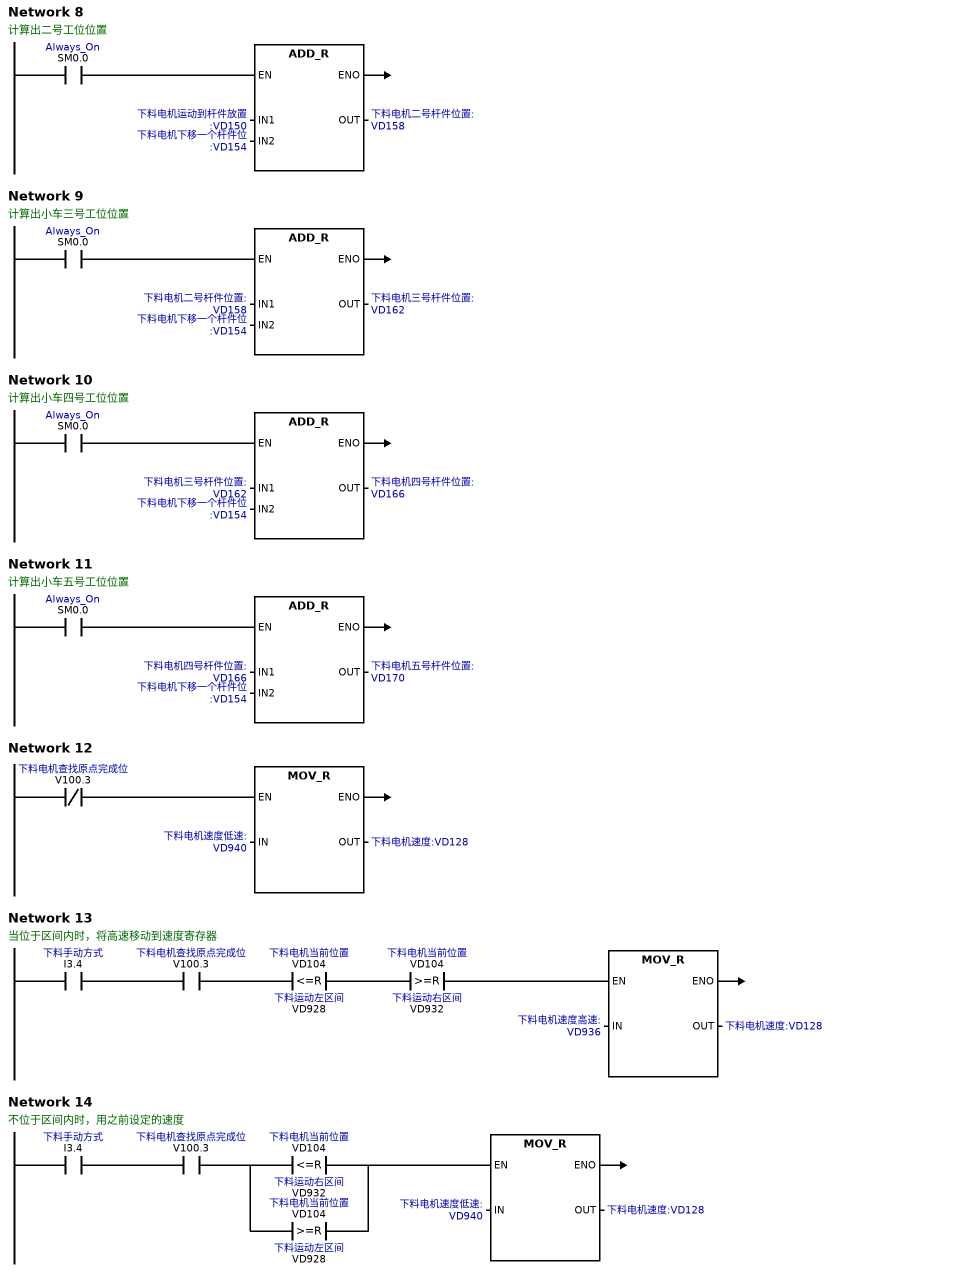
[picture p24: SBR15 networks 8-14]
Network 8
// 计算出二号工位位置
LD     Always_On:SM0.0
MOVR   下料电机运动到杆件放置:VD150, 下料电机二号杆件位置:VD158
+R     下料电机下移一个杆件位:VD154, 下料电机二号杆件位置:VD158
Network 9
// 计算出小车三号工位位置
LD     Always_On:SM0.0
MOVR   下料电机二号杆件位置:VD158, 下料电机三号杆件位置:VD162
+R     下料电机下移一个杆件位:VD154, 下料电机三号杆件位置:VD162
Network 10
// 计算出小车四号工位位置
LD     Always_On:SM0.0
MOVR   下料电机三号杆件位置:VD162, 下料电机四号杆件位置:VD166
+R     下料电机下移一个杆件位:VD154, 下料电机四号杆件位置:VD166
Network 11
// 计算出小车五号工位位置
LD     Always_On:SM0.0
MOVR   下料电机四号杆件位置:VD166, 下料电机五号杆件位置:VD170
+R     下料电机下移一个杆件位:VD154, 下料电机五号杆件位置:VD170
Network 12
LDN    下料电机查找原点完成位:V100.3
MOVR   下料电机速度低速:VD940, 下料电机速度:VD128
Network 13
// 当位于区间内时，将高速移动到速度寄存器
LD     下料手动方式:I3.4
A      下料电机查找原点完成位:V100.3
AR<=   下料电机当前位置:VD104, 下料运动左区间:VD928
AR>=   下料电机当前位置:VD104, 下料运动右区间:VD932
MOVR   下料电机速度高速:VD936, 下料电机速度:VD128
Network 14
// 不位于区间内时，用之前设定的速度
LD     下料手动方式:I3.4
A      下料电机查找原点完成位:V100.3
LDR<=  下料电机当前位置:VD104, 下料运动右区间:VD932
OR>=   下料电机当前位置:VD104, 下料运动左区间:VD928
ALD
MOVR   下料电机速度低速:VD940, 下料电机速度:VD128
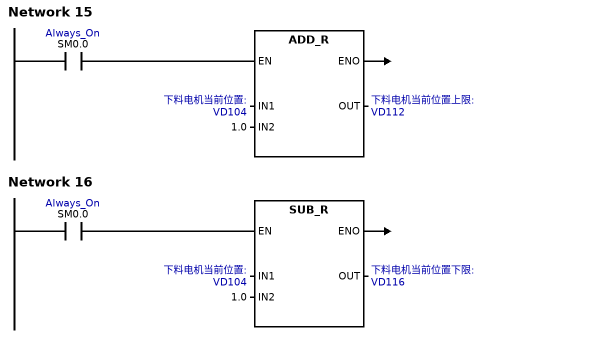
Network 15
LD     Always_On:SM0.0
MOVR   下料电机当前位置:VD104, 下料电机当前位置上限:VD112
+R     1.0, 下料电机当前位置上限:VD112
Network 16
LD     Always_On:SM0.0
MOVR   下料电机当前位置:VD104, 下料电机当前位置下限:VD116
-R     1.0, 下料电机当前位置下限:VD116
END_SUBROUTINE_BLOCK

SUBROUTINE_BLOCK 冷却初始化:SBR16
TITLE=子程序注释
BEGIN
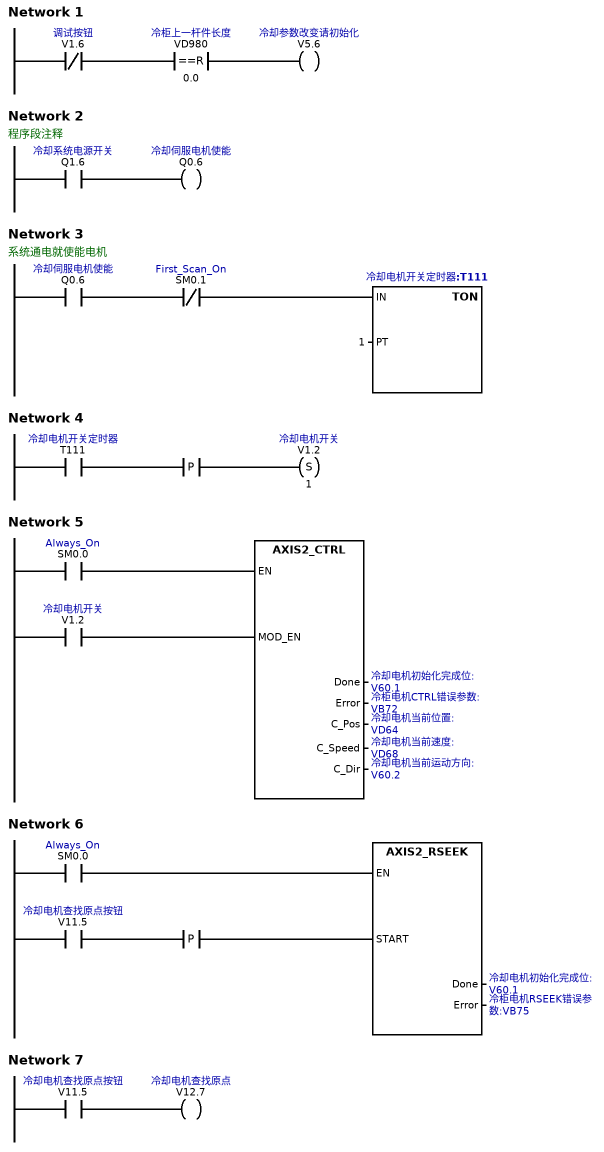
Network 1
LDN    调试按钮:V1.6
AR=    冷柜上一杆件长度:VD980, 0.0
=      冷却参数改变请初始化:V5.6
Network 2
// 程序段注释
LD     冷却系统电源开关:Q1.6
=      冷却伺服电机使能:Q0.6
Network 3
// 系统通电就使能电机
LD     冷却伺服电机使能:Q0.6
AN     First_Scan_On:SM0.1
TON    冷却电机开关定时器:T111, 1
Network 4
LD     冷却电机开关定时器:T111
EU
S      冷却电机开关:V1.2, 1
Network 5
LD     Always_On:SM0.0
=      L60.0
LD     冷却电机开关:V1.2
=      L63.7
LD     L60.0
CALL   AXIS2_CTRL:SBR10, L63.7, 冷却电机初始化完成位:V60.1, 冷柜电机CTRL错误参数:VB72, 冷却电机当前位置:VD64, 冷却电机当前速度:VD68, 冷却电机当前运动方向:V60.2
Network 6
LD     Always_On:SM0.0
=      L60.0
LD     冷却电机查找原点按钮:V11.5
EU
=      L63.7
LD     L60.0
CALL   AXIS2_RSEEK:SBR13, L63.7, 冷却电机初始化完成位:V60.1, 冷柜电机RSEEK错误参数:VB75
Network 7
LD     冷却电机查找原点按钮:V11.5
=      冷却电机查找原点:V12.7
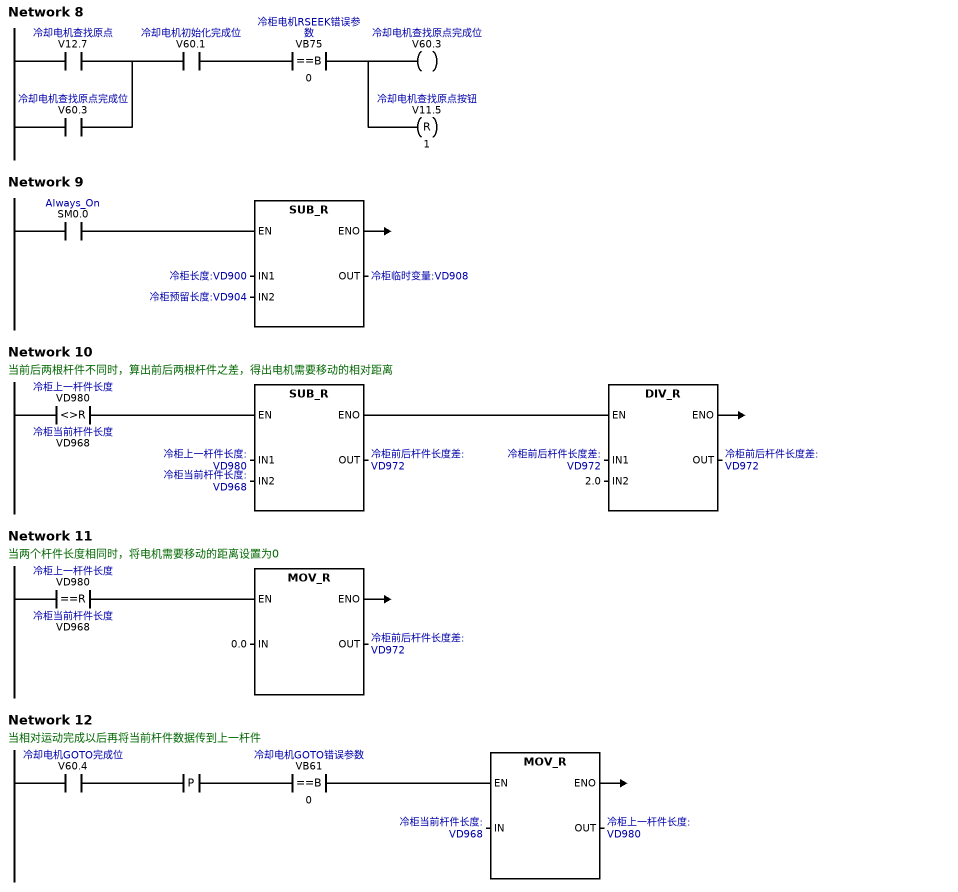
Network 8
LD     冷却电机查找原点:V12.7
O      冷却电机查找原点完成位:V60.3
A      冷却电机初始化完成位:V60.1
AB=    冷柜电机RSEEK错误参数:VB75, 0
=      冷却电机查找原点完成位:V60.3
R      冷却电机查找原点按钮:V11.5, 1
Network 9
LD     Always_On:SM0.0
MOVR   冷柜长度:VD900, 冷柜临时变量:VD908
-R     冷柜预留长度:VD904, 冷柜临时变量:VD908
Network 10
// 当前后两根杆件不同时，算出前后两根杆件之差，得出电机需要移动的相对距离
LDR<>  冷柜上一杆件长度:VD980, 冷柜当前杆件长度:VD968
MOVR   冷柜上一杆件长度:VD980, 冷柜前后杆件长度差:VD972
AENO
-R     冷柜当前杆件长度:VD968, 冷柜前后杆件长度差:VD972
AENO
/R     2.0, 冷柜前后杆件长度差:VD972
Network 11
// 当两个杆件长度相同时，将电机需要移动的距离设置为0
LDR=   冷柜上一杆件长度:VD980, 冷柜当前杆件长度:VD968
MOVR   0.0, 冷柜前后杆件长度差:VD972
Network 12
// 当相对运动完成以后再将当前杆件数据传到上一杆件
LD     冷却电机GOTO完成位:V60.4
EU
AB=    冷却电机GOTO错误参数:VB61, 0
MOVR   冷柜当前杆件长度:VD968, 冷柜上一杆件长度:VD980
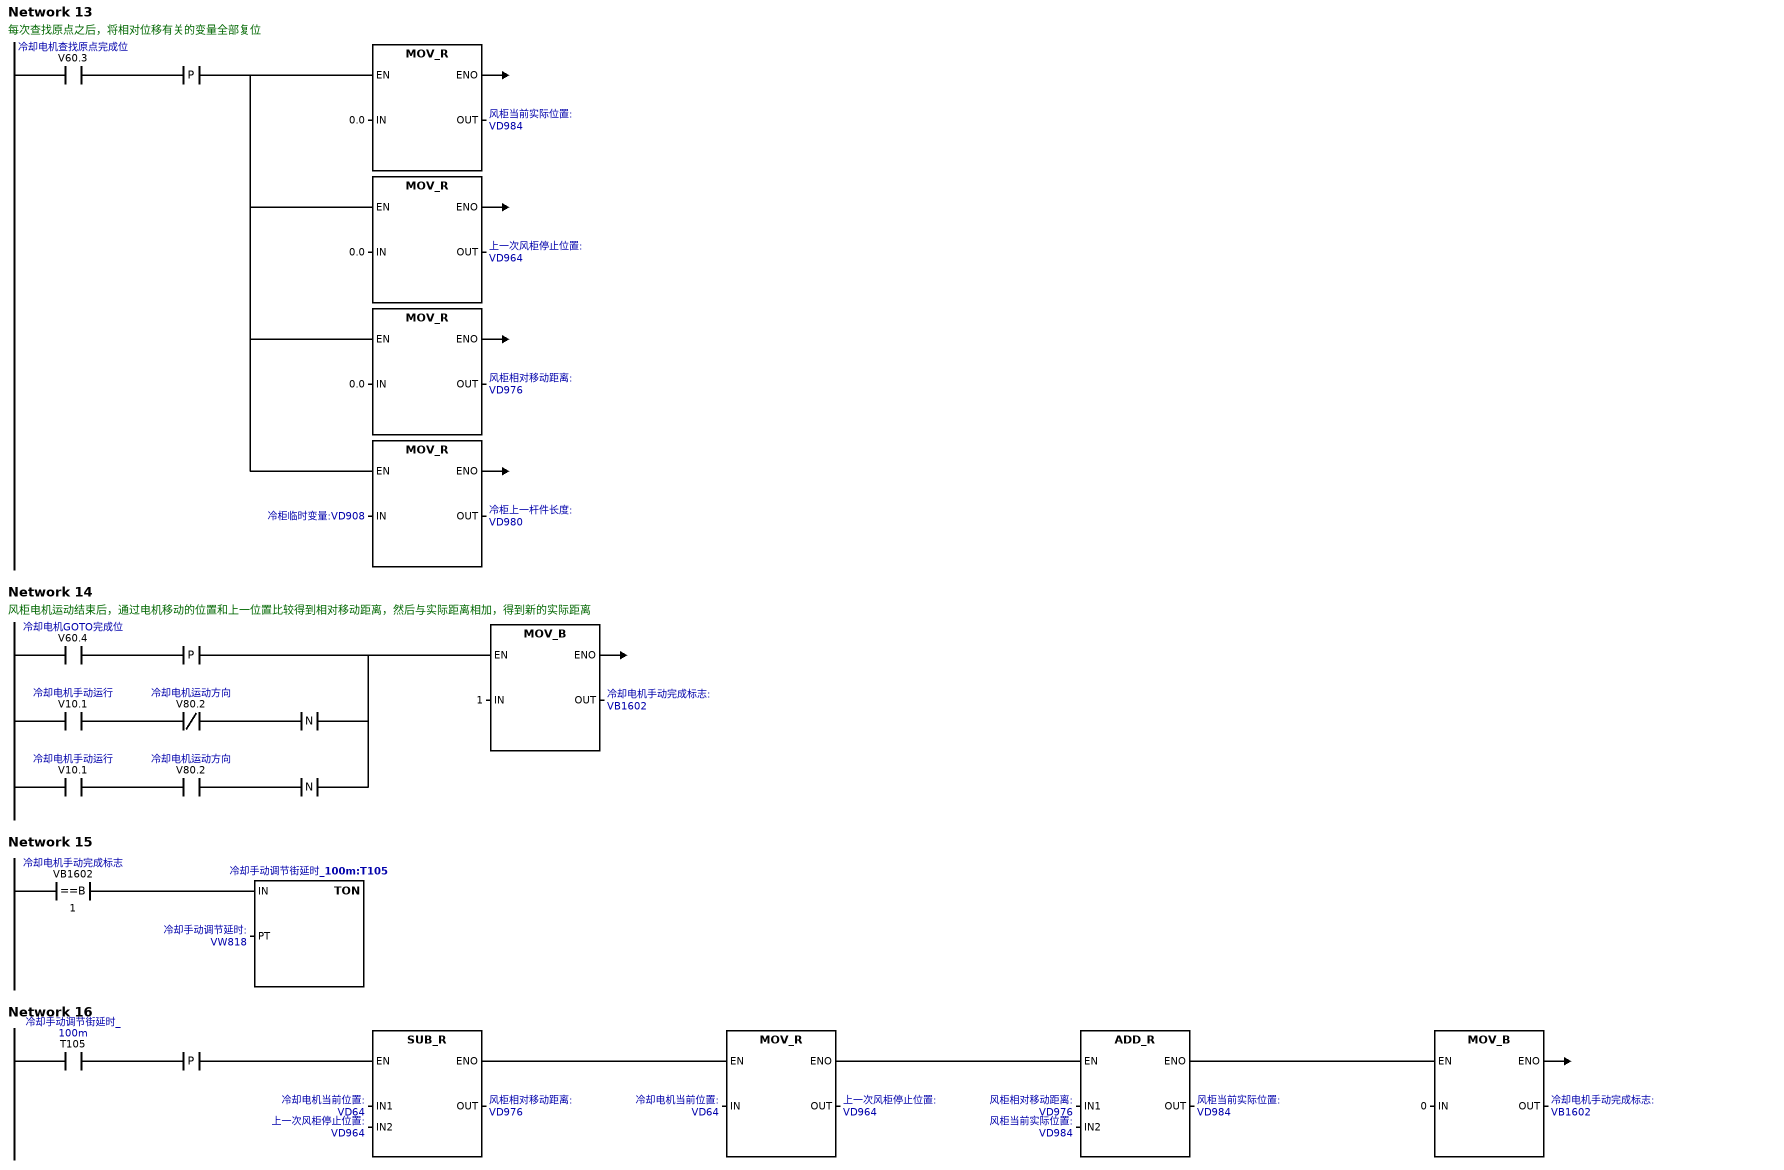
Network 13
// 每次查找原点之后，将相对位移有关的变量全部复位
LD     冷却电机查找原点完成位:V60.3
EU
MOVR   0.0, 风柜当前实际位置:VD984
MOVR   0.0, 上一次风柜停止位置:VD964
MOVR   0.0, 风柜相对移动距离:VD976
MOVR   冷柜临时变量:VD908, 冷柜上一杆件长度:VD980
Network 14
// 风柜电机运动结束后，通过电机移动的位置和上一位置比较得到相对移动距离，然后与实际距离相加，得到新的实际距离
LD     冷却电机GOTO完成位:V60.4
EU
LD     冷却电机手动运行:V10.1
AN     冷却电机运动方向:V80.2
ED
OLD
LD     冷却电机手动运行:V10.1
A      冷却电机运动方向:V80.2
ED
OLD
MOVB   1, 冷却电机手动完成标志:VB1602
Network 15
LDB=   冷却电机手动完成标志:VB1602, 1
TON    冷却手动调节街延时_100m:T105, 冷却手动调节延时:VW818
Network 16
LD     冷却手动调节街延时_100m:T105
EU
MOVR   冷却电机当前位置:VD64, 风柜相对移动距离:VD976
AENO
-R     上一次风柜停止位置:VD964, 风柜相对移动距离:VD976
AENO
MOVR   冷却电机当前位置:VD64, 上一次风柜停止位置:VD964
AENO
+R     风柜相对移动距离:VD976, 风柜当前实际位置:VD984
AENO
MOVB   0, 冷却电机手动完成标志:VB1602
END_SUBROUTINE_BLOCK

SUBROUTINE_BLOCK 上料选号:SBR17
TITLE=子程序注释
BEGIN
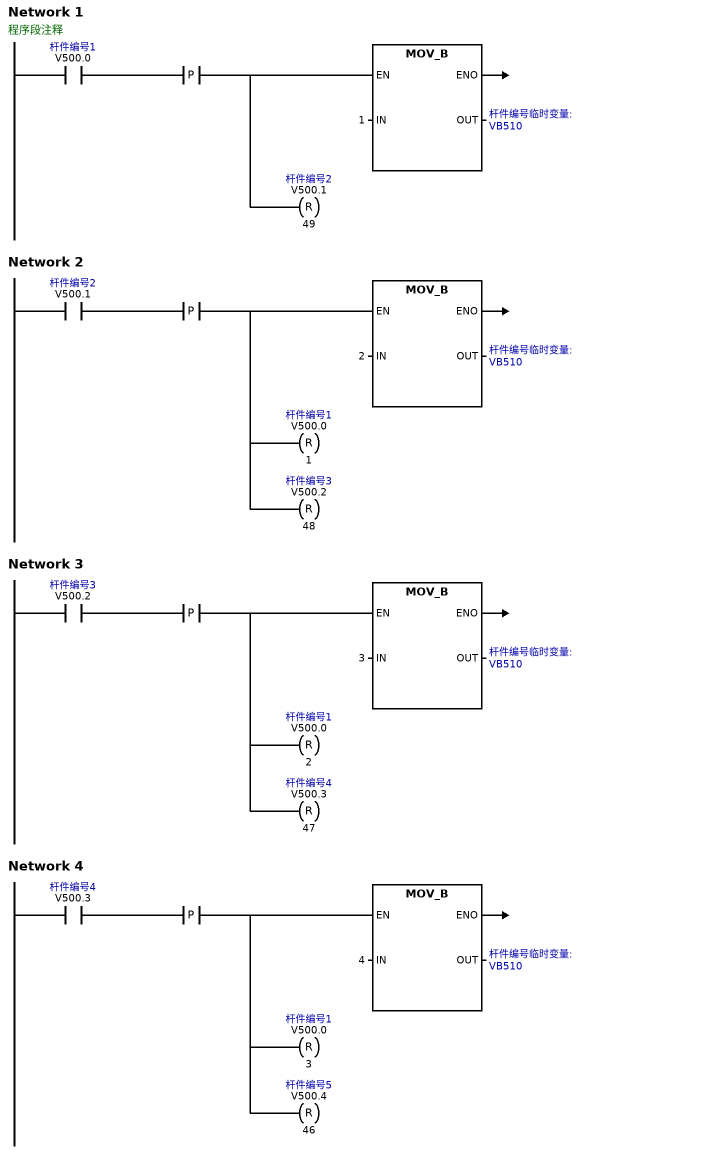
Network 1
// 程序段注释
LD     杆件编号1:V500.0
EU
MOVB   1, 杆件编号临时变量:VB510
R      杆件编号2:V500.1, 49
Network 2
LD     杆件编号2:V500.1
EU
MOVB   2, 杆件编号临时变量:VB510
R      杆件编号1:V500.0, 1
R      杆件编号3:V500.2, 48
Network 3
LD     杆件编号3:V500.2
EU
MOVB   3, 杆件编号临时变量:VB510
R      杆件编号1:V500.0, 2
R      杆件编号4:V500.3, 47
Network 4
LD     杆件编号4:V500.3
EU
MOVB   4, 杆件编号临时变量:VB510
R      杆件编号1:V500.0, 3
R      杆件编号5:V500.4, 46
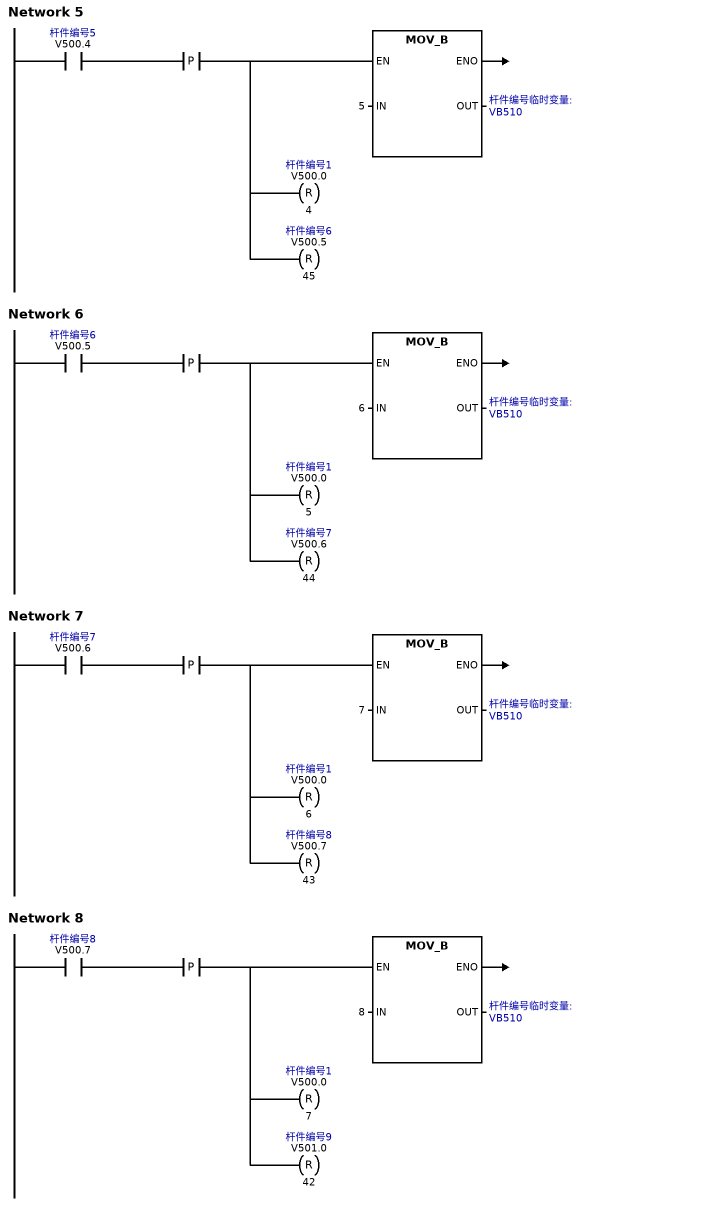
Network 5
LD     杆件编号5:V500.4
EU
MOVB   5, 杆件编号临时变量:VB510
R      杆件编号1:V500.0, 4
R      杆件编号6:V500.5, 45
Network 6
LD     杆件编号6:V500.5
EU
MOVB   6, 杆件编号临时变量:VB510
R      杆件编号1:V500.0, 5
R      杆件编号7:V500.6, 44
Network 7
LD     杆件编号7:V500.6
EU
MOVB   7, 杆件编号临时变量:VB510
R      杆件编号1:V500.0, 6
R      杆件编号8:V500.7, 43
Network 8
LD     杆件编号8:V500.7
EU
MOVB   8, 杆件编号临时变量:VB510
R      杆件编号1:V500.0, 7
R      杆件编号9:V501.0, 42
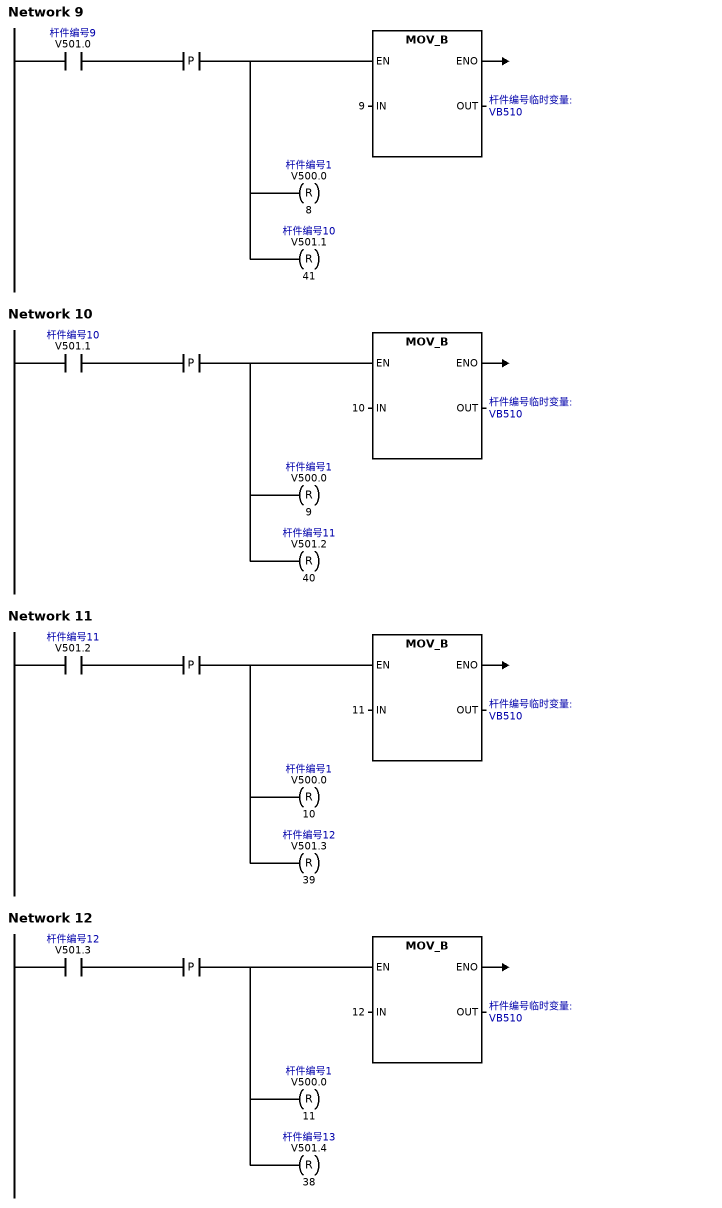
Network 9
LD     杆件编号9:V501.0
EU
MOVB   9, 杆件编号临时变量:VB510
R      杆件编号1:V500.0, 8
R      杆件编号10:V501.1, 41
Network 10
LD     杆件编号10:V501.1
EU
MOVB   10, 杆件编号临时变量:VB510
R      杆件编号1:V500.0, 9
R      杆件编号11:V501.2, 40
Network 11
LD     杆件编号11:V501.2
EU
MOVB   11, 杆件编号临时变量:VB510
R      杆件编号1:V500.0, 10
R      杆件编号12:V501.3, 39
Network 12
LD     杆件编号12:V501.3
EU
MOVB   12, 杆件编号临时变量:VB510
R      杆件编号1:V500.0, 11
R      杆件编号13:V501.4, 38
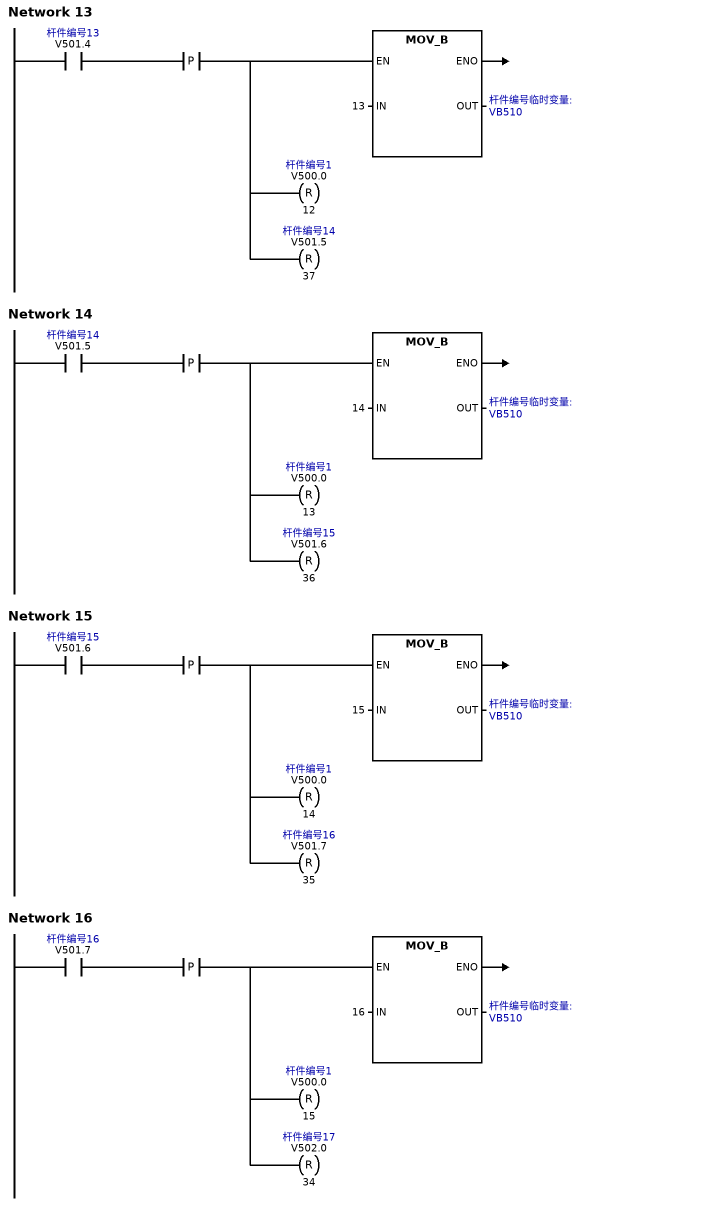
Network 13
LD     杆件编号13:V501.4
EU
MOVB   13, 杆件编号临时变量:VB510
R      杆件编号1:V500.0, 12
R      杆件编号14:V501.5, 37
Network 14
LD     杆件编号14:V501.5
EU
MOVB   14, 杆件编号临时变量:VB510
R      杆件编号1:V500.0, 13
R      杆件编号15:V501.6, 36
Network 15
LD     杆件编号15:V501.6
EU
MOVB   15, 杆件编号临时变量:VB510
R      杆件编号1:V500.0, 14
R      杆件编号16:V501.7, 35
Network 16
LD     杆件编号16:V501.7
EU
MOVB   16, 杆件编号临时变量:VB510
R      杆件编号1:V500.0, 15
R      杆件编号17:V502.0, 34
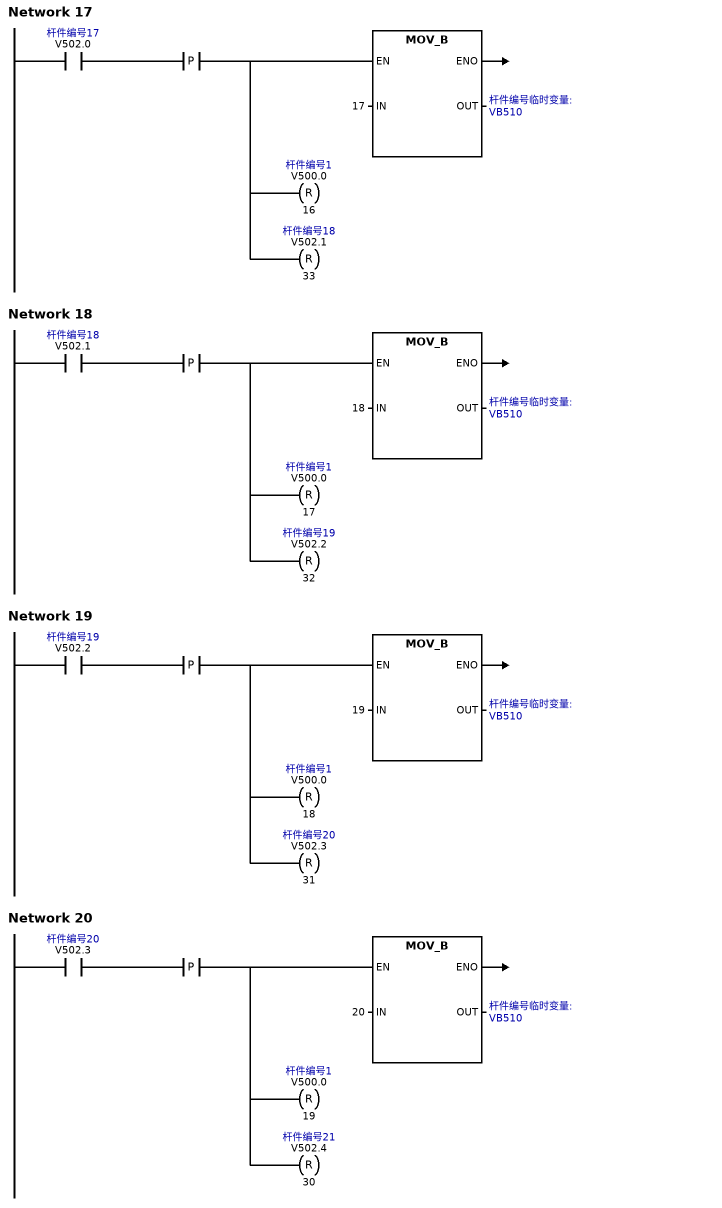
Network 17
LD     杆件编号17:V502.0
EU
MOVB   17, 杆件编号临时变量:VB510
R      杆件编号1:V500.0, 16
R      杆件编号18:V502.1, 33
Network 18
LD     杆件编号18:V502.1
EU
MOVB   18, 杆件编号临时变量:VB510
R      杆件编号1:V500.0, 17
R      杆件编号19:V502.2, 32
Network 19
LD     杆件编号19:V502.2
EU
MOVB   19, 杆件编号临时变量:VB510
R      杆件编号1:V500.0, 18
R      杆件编号20:V502.3, 31
Network 20
LD     杆件编号20:V502.3
EU
MOVB   20, 杆件编号临时变量:VB510
R      杆件编号1:V500.0, 19
R      杆件编号21:V502.4, 30
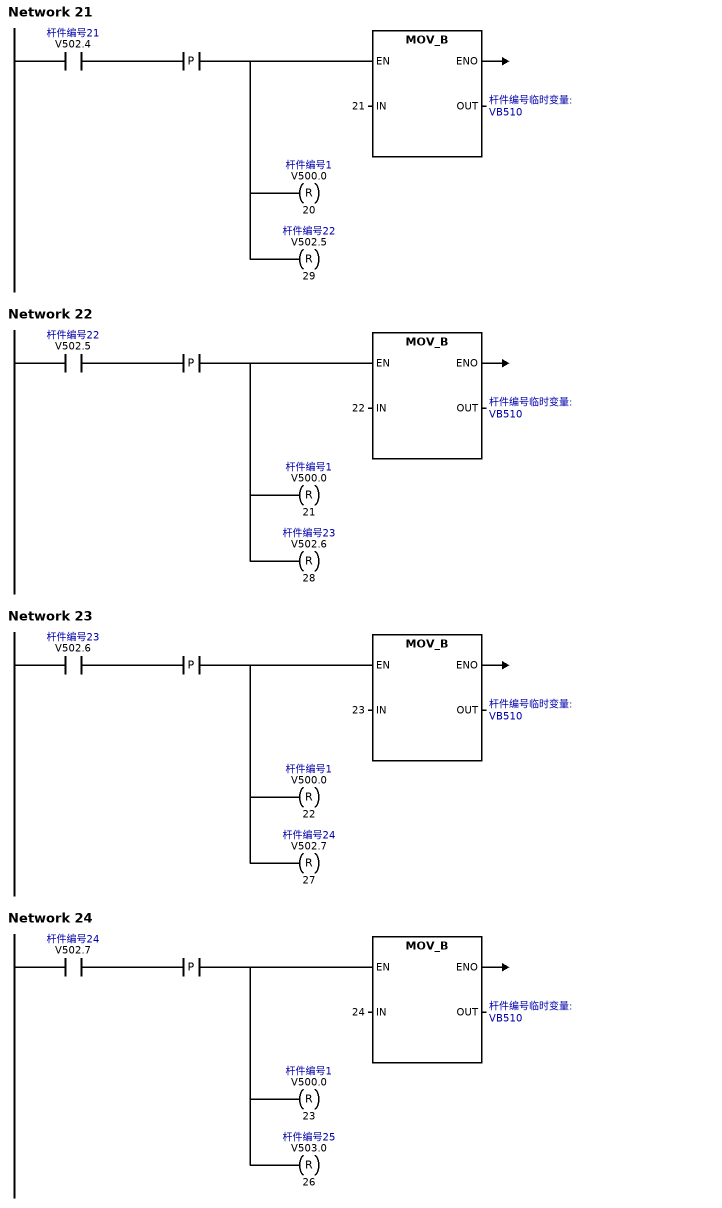
Network 21
LD     杆件编号21:V502.4
EU
MOVB   21, 杆件编号临时变量:VB510
R      杆件编号1:V500.0, 20
R      杆件编号22:V502.5, 29
Network 22
LD     杆件编号22:V502.5
EU
MOVB   22, 杆件编号临时变量:VB510
R      杆件编号1:V500.0, 21
R      杆件编号23:V502.6, 28
Network 23
LD     杆件编号23:V502.6
EU
MOVB   23, 杆件编号临时变量:VB510
R      杆件编号1:V500.0, 22
R      杆件编号24:V502.7, 27
Network 24
LD     杆件编号24:V502.7
EU
MOVB   24, 杆件编号临时变量:VB510
R      杆件编号1:V500.0, 23
R      杆件编号25:V503.0, 26
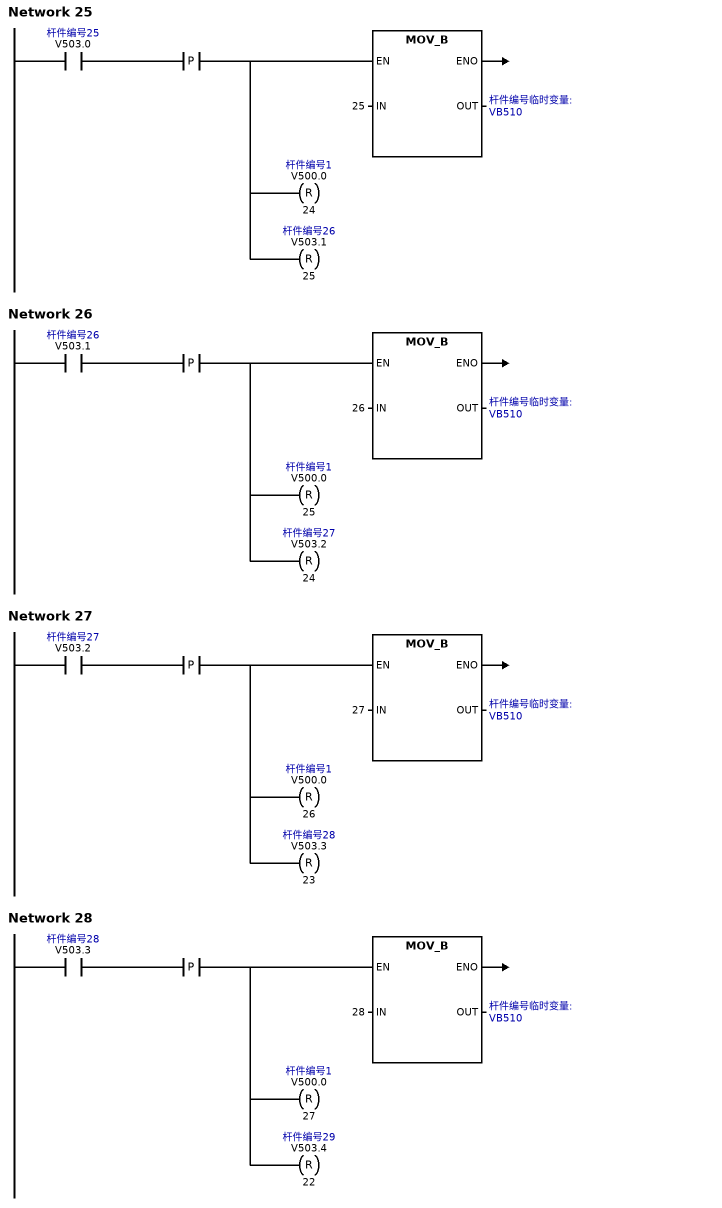
Network 25
LD     杆件编号25:V503.0
EU
MOVB   25, 杆件编号临时变量:VB510
R      杆件编号1:V500.0, 24
R      杆件编号26:V503.1, 25
Network 26
LD     杆件编号26:V503.1
EU
MOVB   26, 杆件编号临时变量:VB510
R      杆件编号1:V500.0, 25
R      杆件编号27:V503.2, 24
Network 27
LD     杆件编号27:V503.2
EU
MOVB   27, 杆件编号临时变量:VB510
R      杆件编号1:V500.0, 26
R      杆件编号28:V503.3, 23
Network 28
LD     杆件编号28:V503.3
EU
MOVB   28, 杆件编号临时变量:VB510
R      杆件编号1:V500.0, 27
R      杆件编号29:V503.4, 22
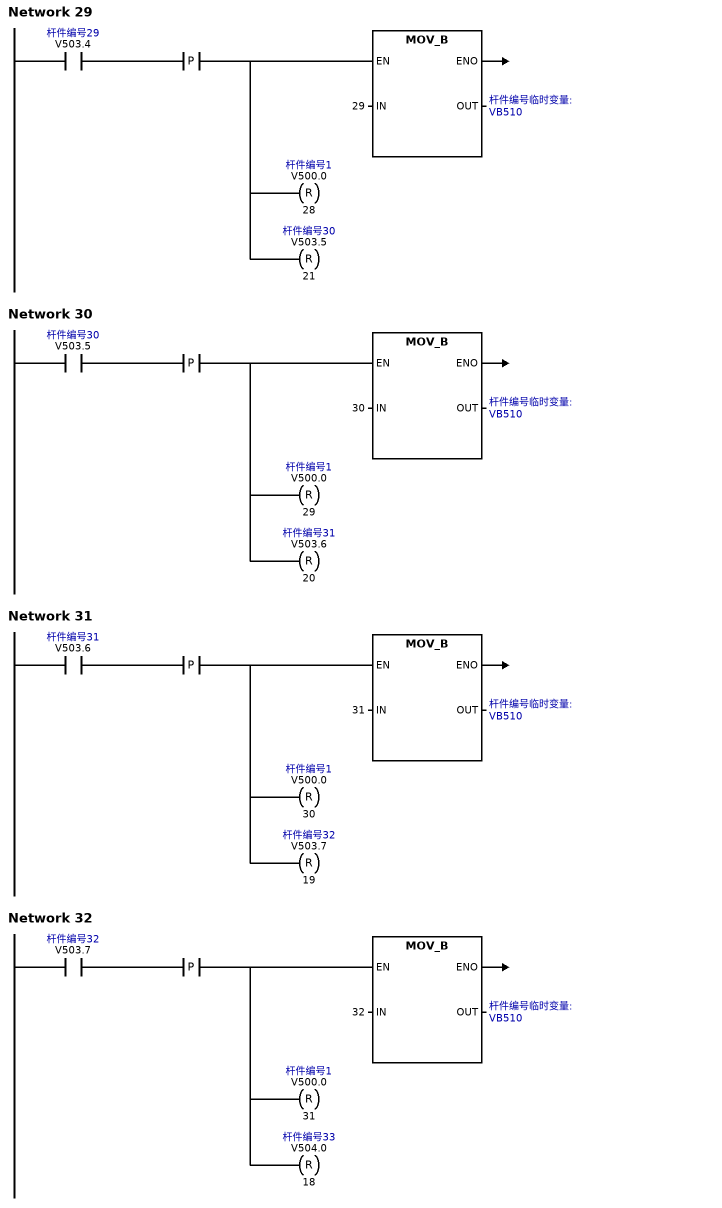
Network 29
LD     杆件编号29:V503.4
EU
MOVB   29, 杆件编号临时变量:VB510
R      杆件编号1:V500.0, 28
R      杆件编号30:V503.5, 21
Network 30
LD     杆件编号30:V503.5
EU
MOVB   30, 杆件编号临时变量:VB510
R      杆件编号1:V500.0, 29
R      杆件编号31:V503.6, 20
Network 31
LD     杆件编号31:V503.6
EU
MOVB   31, 杆件编号临时变量:VB510
R      杆件编号1:V500.0, 30
R      杆件编号32:V503.7, 19
Network 32
LD     杆件编号32:V503.7
EU
MOVB   32, 杆件编号临时变量:VB510
R      杆件编号1:V500.0, 31
R      杆件编号33:V504.0, 18
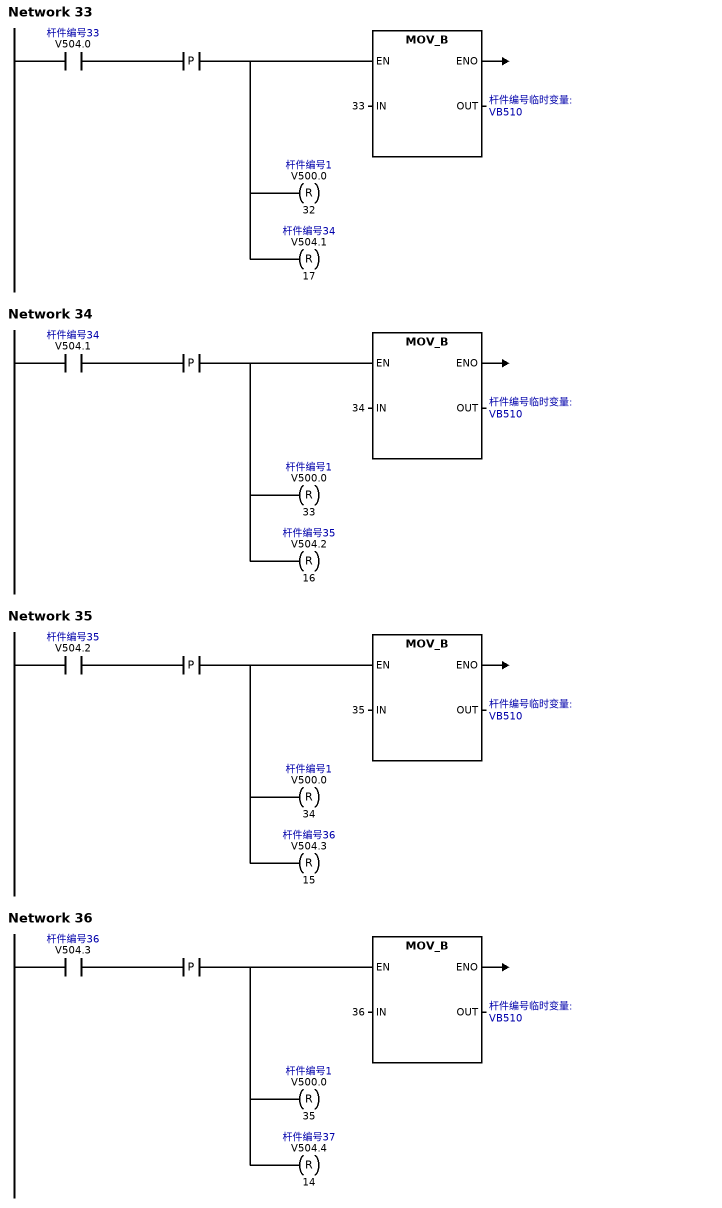
Network 33
LD     杆件编号33:V504.0
EU
MOVB   33, 杆件编号临时变量:VB510
R      杆件编号1:V500.0, 32
R      杆件编号34:V504.1, 17
Network 34
LD     杆件编号34:V504.1
EU
MOVB   34, 杆件编号临时变量:VB510
R      杆件编号1:V500.0, 33
R      杆件编号35:V504.2, 16
Network 35
LD     杆件编号35:V504.2
EU
MOVB   35, 杆件编号临时变量:VB510
R      杆件编号1:V500.0, 34
R      杆件编号36:V504.3, 15
Network 36
LD     杆件编号36:V504.3
EU
MOVB   36, 杆件编号临时变量:VB510
R      杆件编号1:V500.0, 35
R      杆件编号37:V504.4, 14
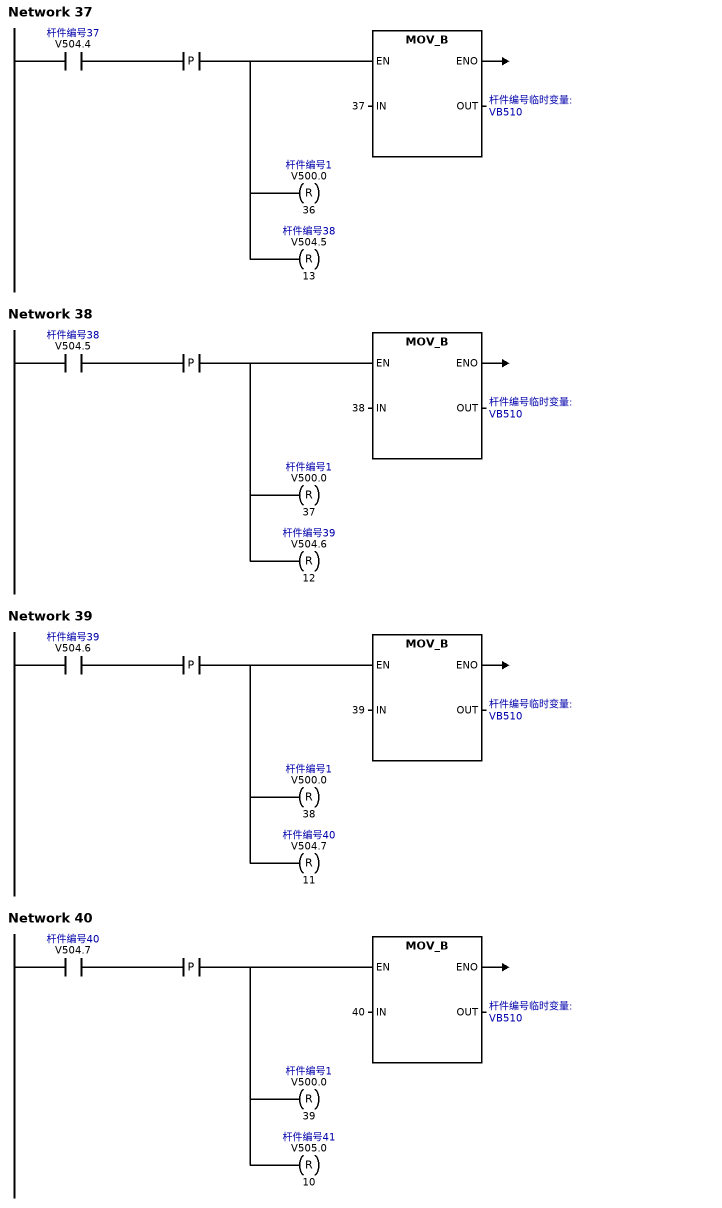
Network 37
LD     杆件编号37:V504.4
EU
MOVB   37, 杆件编号临时变量:VB510
R      杆件编号1:V500.0, 36
R      杆件编号38:V504.5, 13
Network 38
LD     杆件编号38:V504.5
EU
MOVB   38, 杆件编号临时变量:VB510
R      杆件编号1:V500.0, 37
R      杆件编号39:V504.6, 12
Network 39
LD     杆件编号39:V504.6
EU
MOVB   39, 杆件编号临时变量:VB510
R      杆件编号1:V500.0, 38
R      杆件编号40:V504.7, 11
Network 40
LD     杆件编号40:V504.7
EU
MOVB   40, 杆件编号临时变量:VB510
R      杆件编号1:V500.0, 39
R      杆件编号41:V505.0, 10
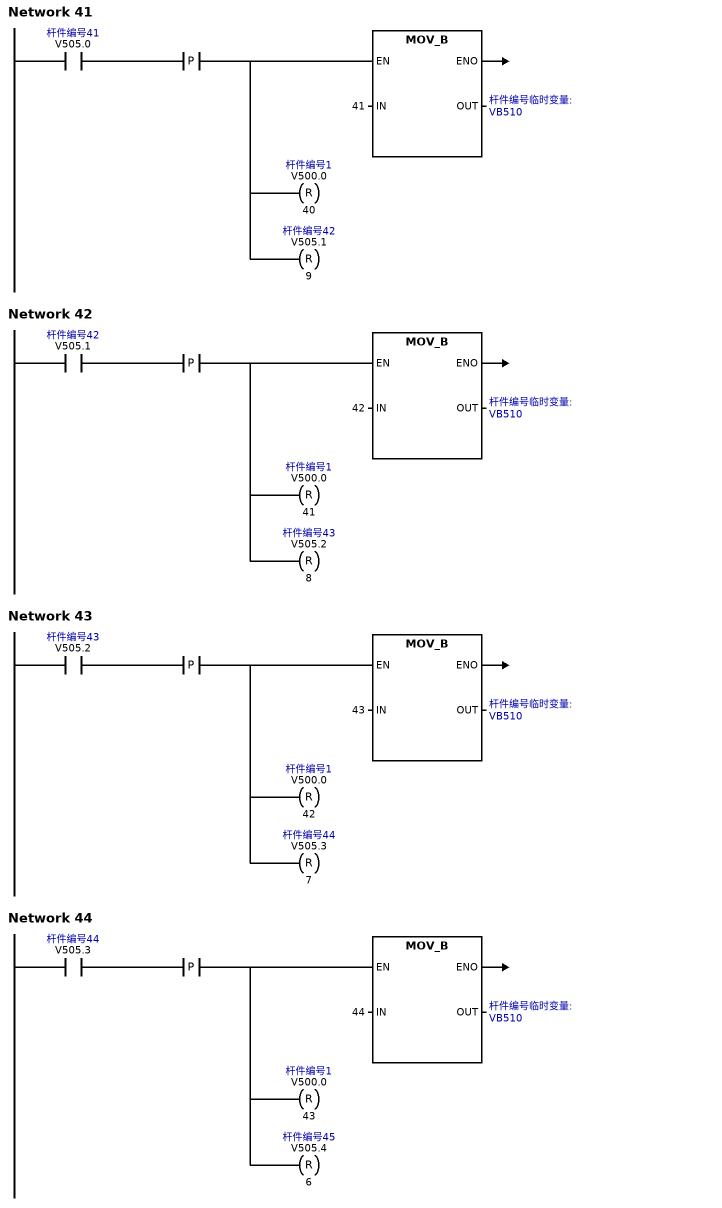
Network 41
LD     杆件编号41:V505.0
EU
MOVB   41, 杆件编号临时变量:VB510
R      杆件编号1:V500.0, 40
R      杆件编号42:V505.1, 9
Network 42
LD     杆件编号42:V505.1
EU
MOVB   42, 杆件编号临时变量:VB510
R      杆件编号1:V500.0, 41
R      杆件编号43:V505.2, 8
Network 43
LD     杆件编号43:V505.2
EU
MOVB   43, 杆件编号临时变量:VB510
R      杆件编号1:V500.0, 42
R      杆件编号44:V505.3, 7
Network 44
LD     杆件编号44:V505.3
EU
MOVB   44, 杆件编号临时变量:VB510
R      杆件编号1:V500.0, 43
R      杆件编号45:V505.4, 6
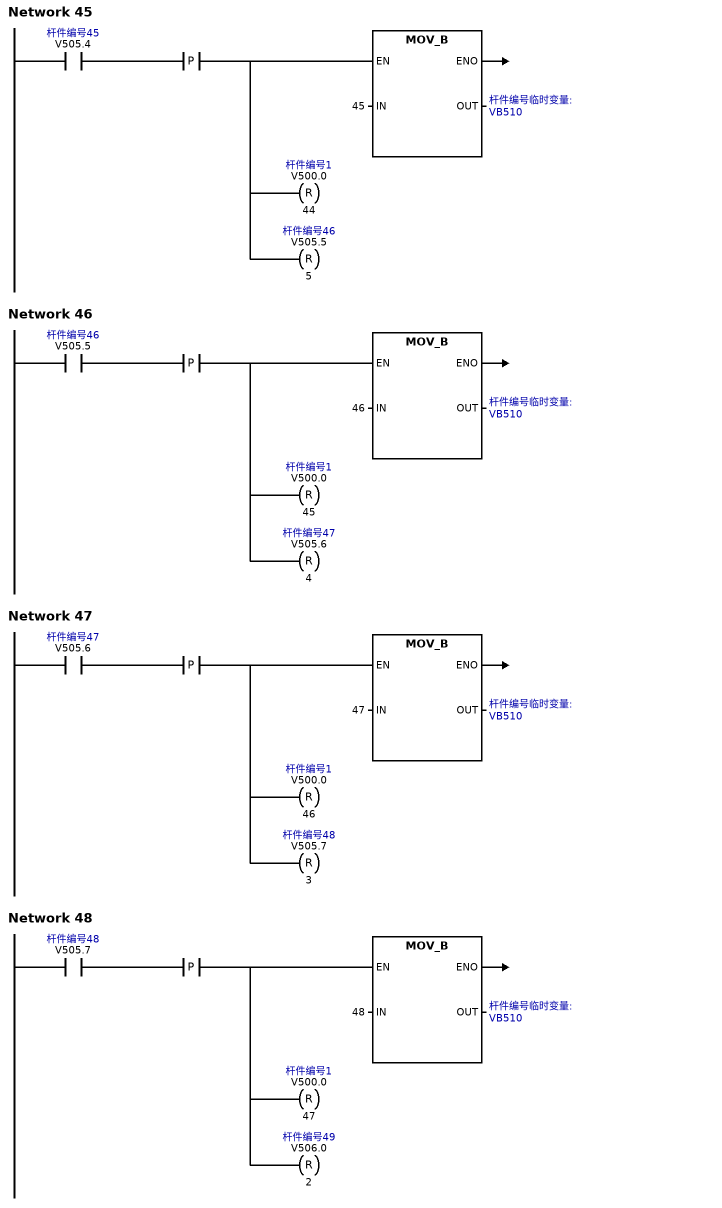
Network 45
LD     杆件编号45:V505.4
EU
MOVB   45, 杆件编号临时变量:VB510
R      杆件编号1:V500.0, 44
R      杆件编号46:V505.5, 5
Network 46
LD     杆件编号46:V505.5
EU
MOVB   46, 杆件编号临时变量:VB510
R      杆件编号1:V500.0, 45
R      杆件编号47:V505.6, 4
Network 47
LD     杆件编号47:V505.6
EU
MOVB   47, 杆件编号临时变量:VB510
R      杆件编号1:V500.0, 46
R      杆件编号48:V505.7, 3
Network 48
LD     杆件编号48:V505.7
EU
MOVB   48, 杆件编号临时变量:VB510
R      杆件编号1:V500.0, 47
R      杆件编号49:V506.0, 2
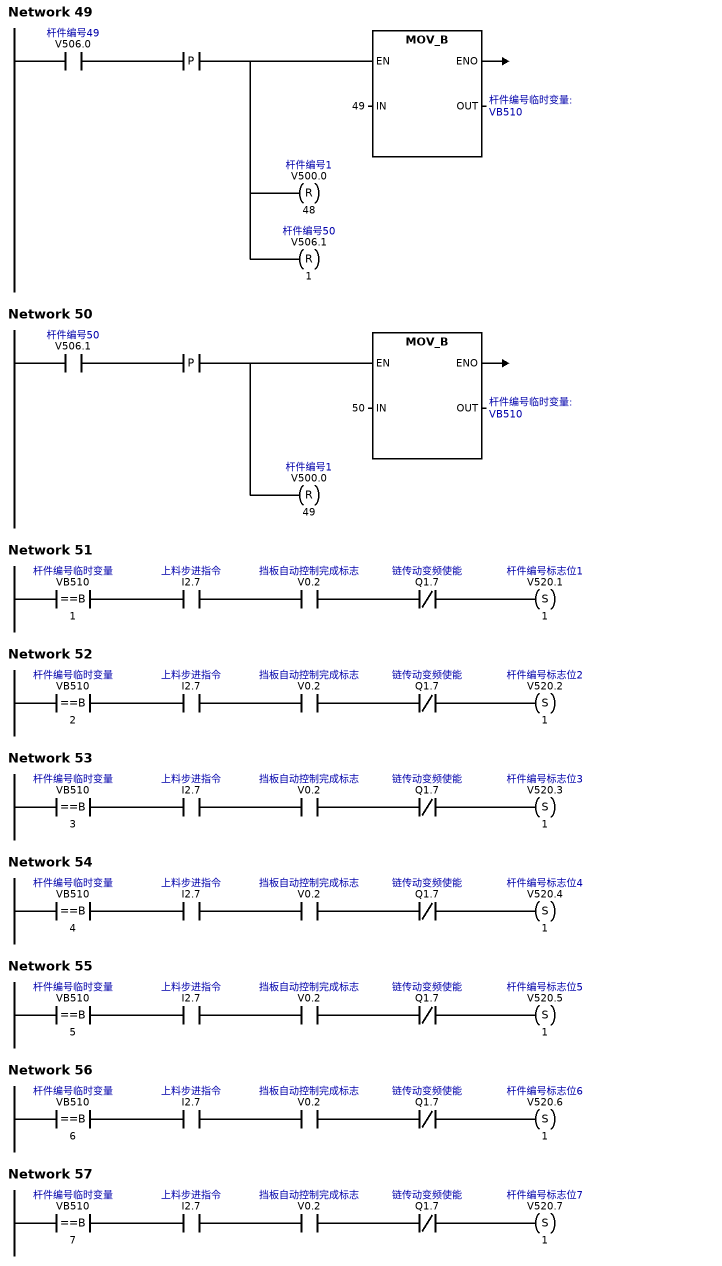
Network 49
LD     杆件编号49:V506.0
EU
MOVB   49, 杆件编号临时变量:VB510
R      杆件编号1:V500.0, 48
R      杆件编号50:V506.1, 1
Network 50
LD     杆件编号50:V506.1
EU
MOVB   50, 杆件编号临时变量:VB510
R      杆件编号1:V500.0, 49
Network 51
LDB=   杆件编号临时变量:VB510, 1
A      上料步进指令:I2.7
A      挡板自动控制完成标志:V0.2
AN     链传动变频使能:Q1.7
S      杆件编号标志位1:V520.1, 1
Network 52
LDB=   杆件编号临时变量:VB510, 2
A      上料步进指令:I2.7
A      挡板自动控制完成标志:V0.2
AN     链传动变频使能:Q1.7
S      杆件编号标志位2:V520.2, 1
Network 53
LDB=   杆件编号临时变量:VB510, 3
A      上料步进指令:I2.7
A      挡板自动控制完成标志:V0.2
AN     链传动变频使能:Q1.7
S      杆件编号标志位3:V520.3, 1
Network 54
LDB=   杆件编号临时变量:VB510, 4
A      上料步进指令:I2.7
A      挡板自动控制完成标志:V0.2
AN     链传动变频使能:Q1.7
S      杆件编号标志位4:V520.4, 1
Network 55
LDB=   杆件编号临时变量:VB510, 5
A      上料步进指令:I2.7
A      挡板自动控制完成标志:V0.2
AN     链传动变频使能:Q1.7
S      杆件编号标志位5:V520.5, 1
Network 56
LDB=   杆件编号临时变量:VB510, 6
A      上料步进指令:I2.7
A      挡板自动控制完成标志:V0.2
AN     链传动变频使能:Q1.7
S      杆件编号标志位6:V520.6, 1
Network 57
LDB=   杆件编号临时变量:VB510, 7
A      上料步进指令:I2.7
A      挡板自动控制完成标志:V0.2
AN     链传动变频使能:Q1.7
S      杆件编号标志位7:V520.7, 1
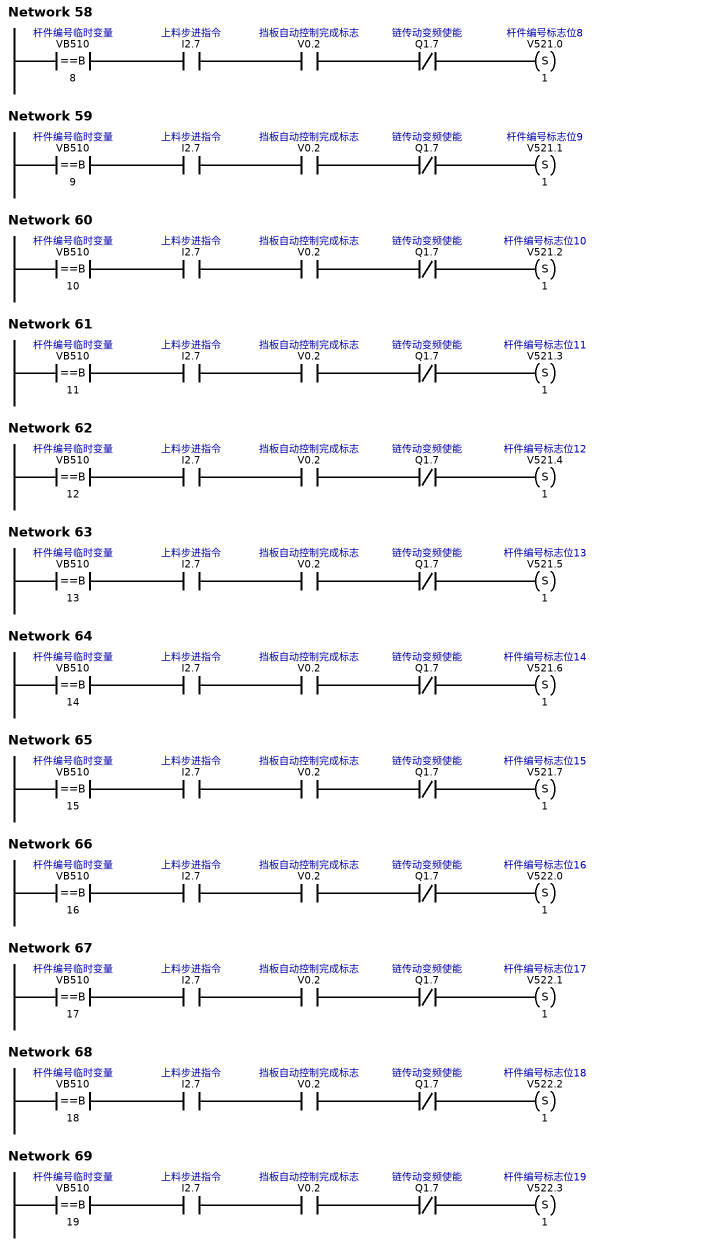
Network 58
LDB=   杆件编号临时变量:VB510, 8
A      上料步进指令:I2.7
A      挡板自动控制完成标志:V0.2
AN     链传动变频使能:Q1.7
S      杆件编号标志位8:V521.0, 1
Network 59
LDB=   杆件编号临时变量:VB510, 9
A      上料步进指令:I2.7
A      挡板自动控制完成标志:V0.2
AN     链传动变频使能:Q1.7
S      杆件编号标志位9:V521.1, 1
Network 60
LDB=   杆件编号临时变量:VB510, 10
A      上料步进指令:I2.7
A      挡板自动控制完成标志:V0.2
AN     链传动变频使能:Q1.7
S      杆件编号标志位10:V521.2, 1
Network 61
LDB=   杆件编号临时变量:VB510, 11
A      上料步进指令:I2.7
A      挡板自动控制完成标志:V0.2
AN     链传动变频使能:Q1.7
S      杆件编号标志位11:V521.3, 1
Network 62
LDB=   杆件编号临时变量:VB510, 12
A      上料步进指令:I2.7
A      挡板自动控制完成标志:V0.2
AN     链传动变频使能:Q1.7
S      杆件编号标志位12:V521.4, 1
Network 63
LDB=   杆件编号临时变量:VB510, 13
A      上料步进指令:I2.7
A      挡板自动控制完成标志:V0.2
AN     链传动变频使能:Q1.7
S      杆件编号标志位13:V521.5, 1
Network 64
LDB=   杆件编号临时变量:VB510, 14
A      上料步进指令:I2.7
A      挡板自动控制完成标志:V0.2
AN     链传动变频使能:Q1.7
S      杆件编号标志位14:V521.6, 1
Network 65
LDB=   杆件编号临时变量:VB510, 15
A      上料步进指令:I2.7
A      挡板自动控制完成标志:V0.2
AN     链传动变频使能:Q1.7
S      杆件编号标志位15:V521.7, 1
Network 66
LDB=   杆件编号临时变量:VB510, 16
A      上料步进指令:I2.7
A      挡板自动控制完成标志:V0.2
AN     链传动变频使能:Q1.7
S      杆件编号标志位16:V522.0, 1
Network 67
LDB=   杆件编号临时变量:VB510, 17
A      上料步进指令:I2.7
A      挡板自动控制完成标志:V0.2
AN     链传动变频使能:Q1.7
S      杆件编号标志位17:V522.1, 1
Network 68
LDB=   杆件编号临时变量:VB510, 18
A      上料步进指令:I2.7
A      挡板自动控制完成标志:V0.2
AN     链传动变频使能:Q1.7
S      杆件编号标志位18:V522.2, 1
Network 69
LDB=   杆件编号临时变量:VB510, 19
A      上料步进指令:I2.7
A      挡板自动控制完成标志:V0.2
AN     链传动变频使能:Q1.7
S      杆件编号标志位19:V522.3, 1
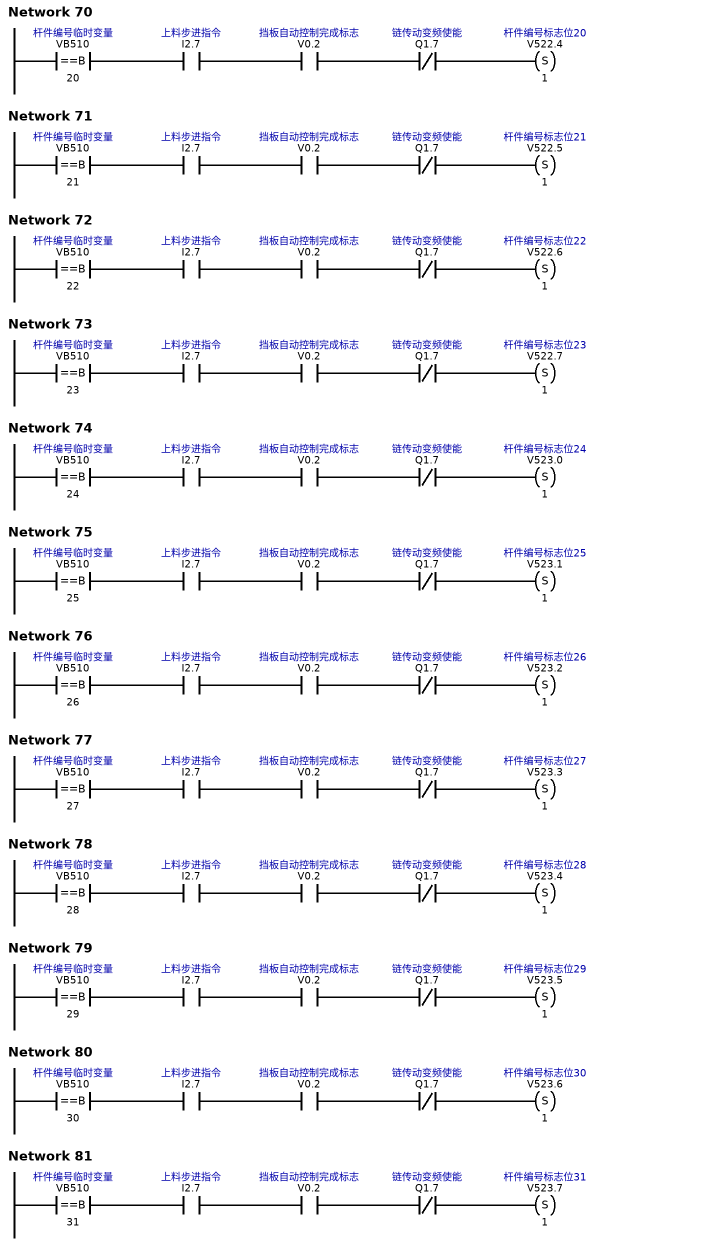
Network 70
LDB=   杆件编号临时变量:VB510, 20
A      上料步进指令:I2.7
A      挡板自动控制完成标志:V0.2
AN     链传动变频使能:Q1.7
S      杆件编号标志位20:V522.4, 1
Network 71
LDB=   杆件编号临时变量:VB510, 21
A      上料步进指令:I2.7
A      挡板自动控制完成标志:V0.2
AN     链传动变频使能:Q1.7
S      杆件编号标志位21:V522.5, 1
Network 72
LDB=   杆件编号临时变量:VB510, 22
A      上料步进指令:I2.7
A      挡板自动控制完成标志:V0.2
AN     链传动变频使能:Q1.7
S      杆件编号标志位22:V522.6, 1
Network 73
LDB=   杆件编号临时变量:VB510, 23
A      上料步进指令:I2.7
A      挡板自动控制完成标志:V0.2
AN     链传动变频使能:Q1.7
S      杆件编号标志位23:V522.7, 1
Network 74
LDB=   杆件编号临时变量:VB510, 24
A      上料步进指令:I2.7
A      挡板自动控制完成标志:V0.2
AN     链传动变频使能:Q1.7
S      杆件编号标志位24:V523.0, 1
Network 75
LDB=   杆件编号临时变量:VB510, 25
A      上料步进指令:I2.7
A      挡板自动控制完成标志:V0.2
AN     链传动变频使能:Q1.7
S      杆件编号标志位25:V523.1, 1
Network 76
LDB=   杆件编号临时变量:VB510, 26
A      上料步进指令:I2.7
A      挡板自动控制完成标志:V0.2
AN     链传动变频使能:Q1.7
S      杆件编号标志位26:V523.2, 1
Network 77
LDB=   杆件编号临时变量:VB510, 27
A      上料步进指令:I2.7
A      挡板自动控制完成标志:V0.2
AN     链传动变频使能:Q1.7
S      杆件编号标志位27:V523.3, 1
Network 78
LDB=   杆件编号临时变量:VB510, 28
A      上料步进指令:I2.7
A      挡板自动控制完成标志:V0.2
AN     链传动变频使能:Q1.7
S      杆件编号标志位28:V523.4, 1
Network 79
LDB=   杆件编号临时变量:VB510, 29
A      上料步进指令:I2.7
A      挡板自动控制完成标志:V0.2
AN     链传动变频使能:Q1.7
S      杆件编号标志位29:V523.5, 1
Network 80
LDB=   杆件编号临时变量:VB510, 30
A      上料步进指令:I2.7
A      挡板自动控制完成标志:V0.2
AN     链传动变频使能:Q1.7
S      杆件编号标志位30:V523.6, 1
Network 81
LDB=   杆件编号临时变量:VB510, 31
A      上料步进指令:I2.7
A      挡板自动控制完成标志:V0.2
AN     链传动变频使能:Q1.7
S      杆件编号标志位31:V523.7, 1
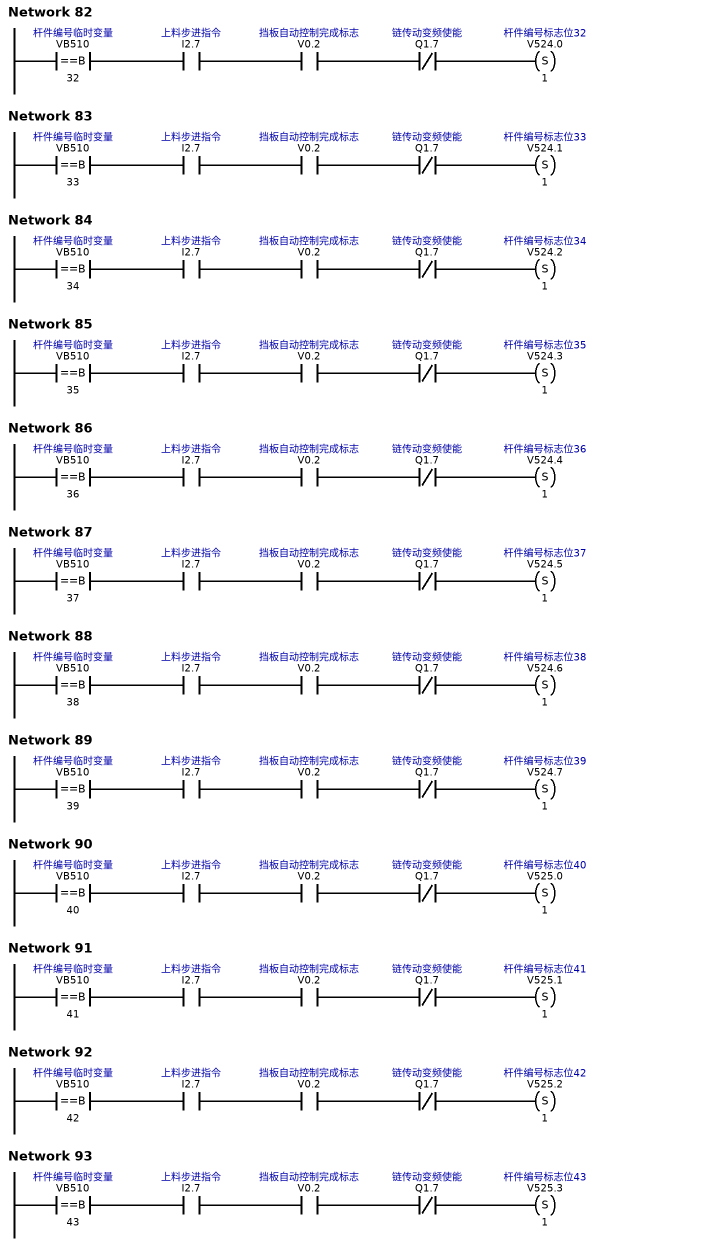
Network 82
LDB=   杆件编号临时变量:VB510, 32
A      上料步进指令:I2.7
A      挡板自动控制完成标志:V0.2
AN     链传动变频使能:Q1.7
S      杆件编号标志位32:V524.0, 1
Network 83
LDB=   杆件编号临时变量:VB510, 33
A      上料步进指令:I2.7
A      挡板自动控制完成标志:V0.2
AN     链传动变频使能:Q1.7
S      杆件编号标志位33:V524.1, 1
Network 84
LDB=   杆件编号临时变量:VB510, 34
A      上料步进指令:I2.7
A      挡板自动控制完成标志:V0.2
AN     链传动变频使能:Q1.7
S      杆件编号标志位34:V524.2, 1
Network 85
LDB=   杆件编号临时变量:VB510, 35
A      上料步进指令:I2.7
A      挡板自动控制完成标志:V0.2
AN     链传动变频使能:Q1.7
S      杆件编号标志位35:V524.3, 1
Network 86
LDB=   杆件编号临时变量:VB510, 36
A      上料步进指令:I2.7
A      挡板自动控制完成标志:V0.2
AN     链传动变频使能:Q1.7
S      杆件编号标志位36:V524.4, 1
Network 87
LDB=   杆件编号临时变量:VB510, 37
A      上料步进指令:I2.7
A      挡板自动控制完成标志:V0.2
AN     链传动变频使能:Q1.7
S      杆件编号标志位37:V524.5, 1
Network 88
LDB=   杆件编号临时变量:VB510, 38
A      上料步进指令:I2.7
A      挡板自动控制完成标志:V0.2
AN     链传动变频使能:Q1.7
S      杆件编号标志位38:V524.6, 1
Network 89
LDB=   杆件编号临时变量:VB510, 39
A      上料步进指令:I2.7
A      挡板自动控制完成标志:V0.2
AN     链传动变频使能:Q1.7
S      杆件编号标志位39:V524.7, 1
Network 90
LDB=   杆件编号临时变量:VB510, 40
A      上料步进指令:I2.7
A      挡板自动控制完成标志:V0.2
AN     链传动变频使能:Q1.7
S      杆件编号标志位40:V525.0, 1
Network 91
LDB=   杆件编号临时变量:VB510, 41
A      上料步进指令:I2.7
A      挡板自动控制完成标志:V0.2
AN     链传动变频使能:Q1.7
S      杆件编号标志位41:V525.1, 1
Network 92
LDB=   杆件编号临时变量:VB510, 42
A      上料步进指令:I2.7
A      挡板自动控制完成标志:V0.2
AN     链传动变频使能:Q1.7
S      杆件编号标志位42:V525.2, 1
Network 93
LDB=   杆件编号临时变量:VB510, 43
A      上料步进指令:I2.7
A      挡板自动控制完成标志:V0.2
AN     链传动变频使能:Q1.7
S      杆件编号标志位43:V525.3, 1
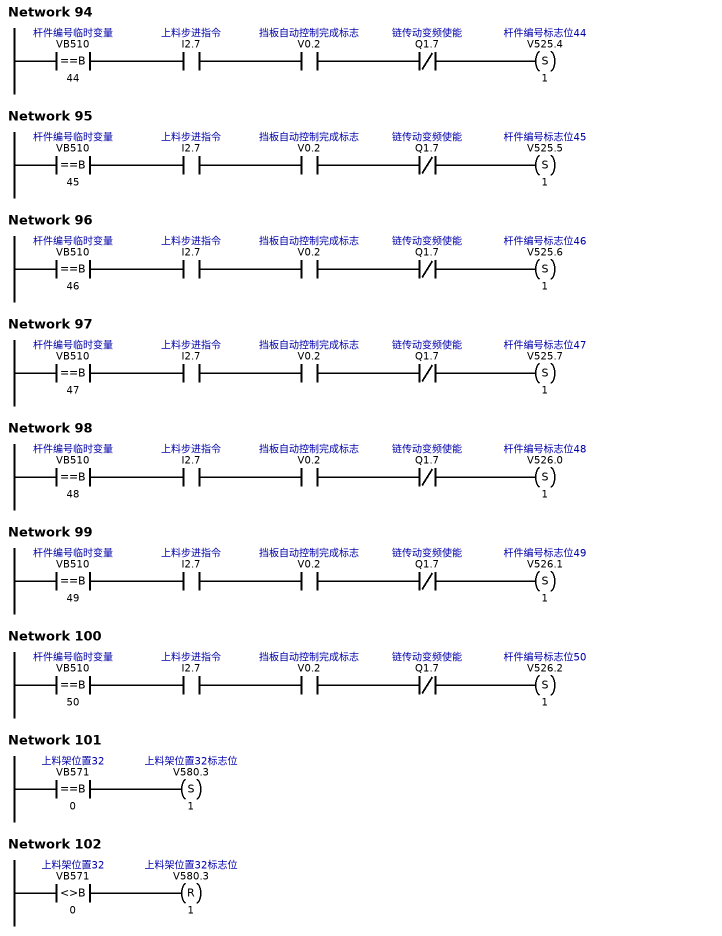
Network 94
LDB=   杆件编号临时变量:VB510, 44
A      上料步进指令:I2.7
A      挡板自动控制完成标志:V0.2
AN     链传动变频使能:Q1.7
S      杆件编号标志位44:V525.4, 1
Network 95
LDB=   杆件编号临时变量:VB510, 45
A      上料步进指令:I2.7
A      挡板自动控制完成标志:V0.2
AN     链传动变频使能:Q1.7
S      杆件编号标志位45:V525.5, 1
Network 96
LDB=   杆件编号临时变量:VB510, 46
A      上料步进指令:I2.7
A      挡板自动控制完成标志:V0.2
AN     链传动变频使能:Q1.7
S      杆件编号标志位46:V525.6, 1
Network 97
LDB=   杆件编号临时变量:VB510, 47
A      上料步进指令:I2.7
A      挡板自动控制完成标志:V0.2
AN     链传动变频使能:Q1.7
S      杆件编号标志位47:V525.7, 1
Network 98
LDB=   杆件编号临时变量:VB510, 48
A      上料步进指令:I2.7
A      挡板自动控制完成标志:V0.2
AN     链传动变频使能:Q1.7
S      杆件编号标志位48:V526.0, 1
Network 99
LDB=   杆件编号临时变量:VB510, 49
A      上料步进指令:I2.7
A      挡板自动控制完成标志:V0.2
AN     链传动变频使能:Q1.7
S      杆件编号标志位49:V526.1, 1
Network 100
LDB=   杆件编号临时变量:VB510, 50
A      上料步进指令:I2.7
A      挡板自动控制完成标志:V0.2
AN     链传动变频使能:Q1.7
S      杆件编号标志位50:V526.2, 1
Network 101
LDB=   上料架位置32:VB571, 0
S      上料架位置32标志位:V580.3, 1
Network 102
LDB<>  上料架位置32:VB571, 0
R      上料架位置32标志位:V580.3, 1
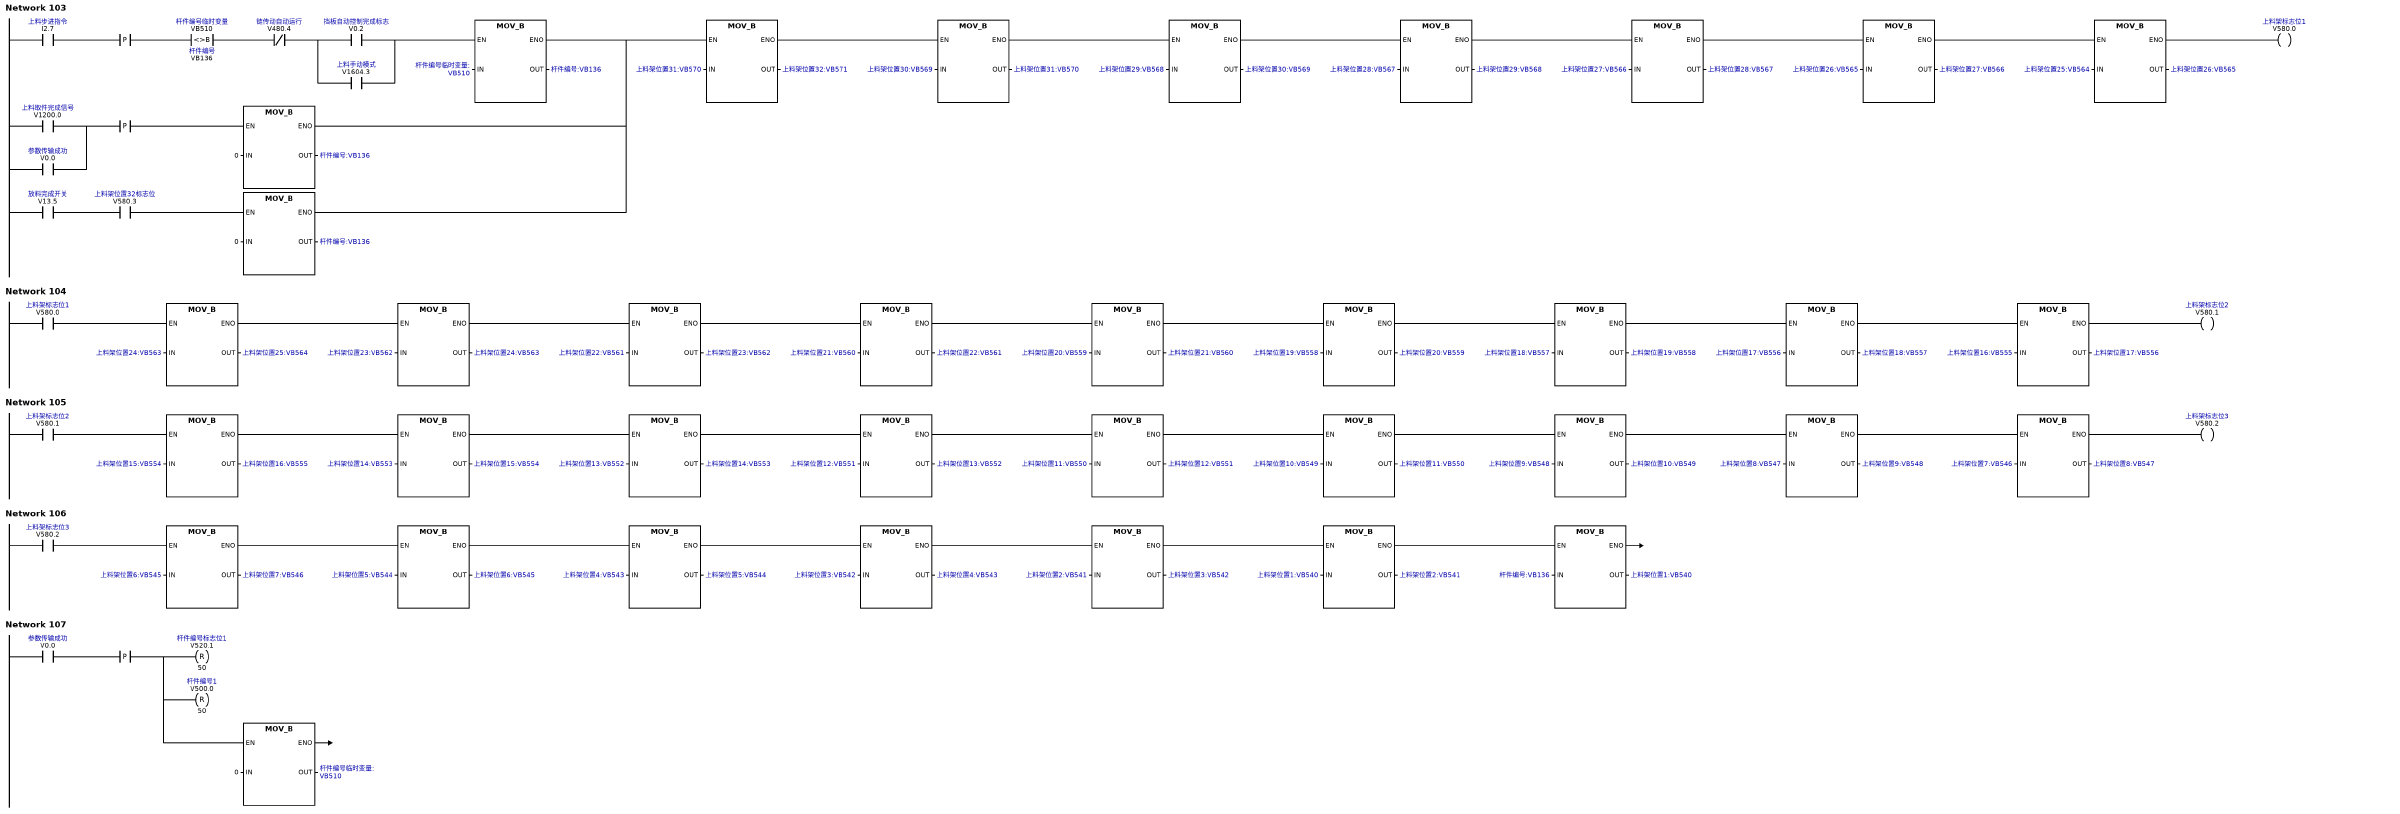
Network 103
LD     上料步进指令:I2.7
EU
AB<>   杆件编号临时变量:VB510, 杆件编号:VB136
AN     链传动自动运行:V480.4
LD     挡板自动控制完成标志:V0.2
O      上料手动模式:V1604.3
ALD
MOVB   杆件编号临时变量:VB510, 杆件编号:VB136
AENO
LD     上料取件完成信号:V1200.0
O      参数传输成功:V0.0
EU
MOVB   0, 杆件编号:VB136
AENO
OLD
LD     放料完成开关:V13.5
A      上料架位置32标志位:V580.3
MOVB   0, 杆件编号:VB136
AENO
OLD
MOVB   上料架位置31:VB570, 上料架位置32:VB571
AENO
MOVB   上料架位置30:VB569, 上料架位置31:VB570
AENO
MOVB   上料架位置29:VB568, 上料架位置30:VB569
AENO
MOVB   上料架位置28:VB567, 上料架位置29:VB568
AENO
MOVB   上料架位置27:VB566, 上料架位置28:VB567
AENO
MOVB   上料架位置26:VB565, 上料架位置27:VB566
AENO
MOVB   上料架位置25:VB564, 上料架位置26:VB565
AENO
=      上料架标志位1:V580.0
Network 104
LD     上料架标志位1:V580.0
MOVB   上料架位置24:VB563, 上料架位置25:VB564
AENO
MOVB   上料架位置23:VB562, 上料架位置24:VB563
AENO
MOVB   上料架位置22:VB561, 上料架位置23:VB562
AENO
MOVB   上料架位置21:VB560, 上料架位置22:VB561
AENO
MOVB   上料架位置20:VB559, 上料架位置21:VB560
AENO
MOVB   上料架位置19:VB558, 上料架位置20:VB559
AENO
MOVB   上料架位置18:VB557, 上料架位置19:VB558
AENO
MOVB   上料架位置17:VB556, 上料架位置18:VB557
AENO
MOVB   上料架位置16:VB555, 上料架位置17:VB556
AENO
=      上料架标志位2:V580.1
Network 105
LD     上料架标志位2:V580.1
MOVB   上料架位置15:VB554, 上料架位置16:VB555
AENO
MOVB   上料架位置14:VB553, 上料架位置15:VB554
AENO
MOVB   上料架位置13:VB552, 上料架位置14:VB553
AENO
MOVB   上料架位置12:VB551, 上料架位置13:VB552
AENO
MOVB   上料架位置11:VB550, 上料架位置12:VB551
AENO
MOVB   上料架位置10:VB549, 上料架位置11:VB550
AENO
MOVB   上料架位置9:VB548, 上料架位置10:VB549
AENO
MOVB   上料架位置8:VB547, 上料架位置9:VB548
AENO
MOVB   上料架位置7:VB546, 上料架位置8:VB547
AENO
=      上料架标志位3:V580.2
Network 106
LD     上料架标志位3:V580.2
MOVB   上料架位置6:VB545, 上料架位置7:VB546
AENO
MOVB   上料架位置5:VB544, 上料架位置6:VB545
AENO
MOVB   上料架位置4:VB543, 上料架位置5:VB544
AENO
MOVB   上料架位置3:VB542, 上料架位置4:VB543
AENO
MOVB   上料架位置2:VB541, 上料架位置3:VB542
AENO
MOVB   上料架位置1:VB540, 上料架位置2:VB541
AENO
MOVB   杆件编号:VB136, 上料架位置1:VB540
Network 107
LD     参数传输成功:V0.0
EU
R      杆件编号标志位1:V520.1, 50
R      杆件编号1:V500.0, 50
MOVB   0, 杆件编号临时变量:VB510
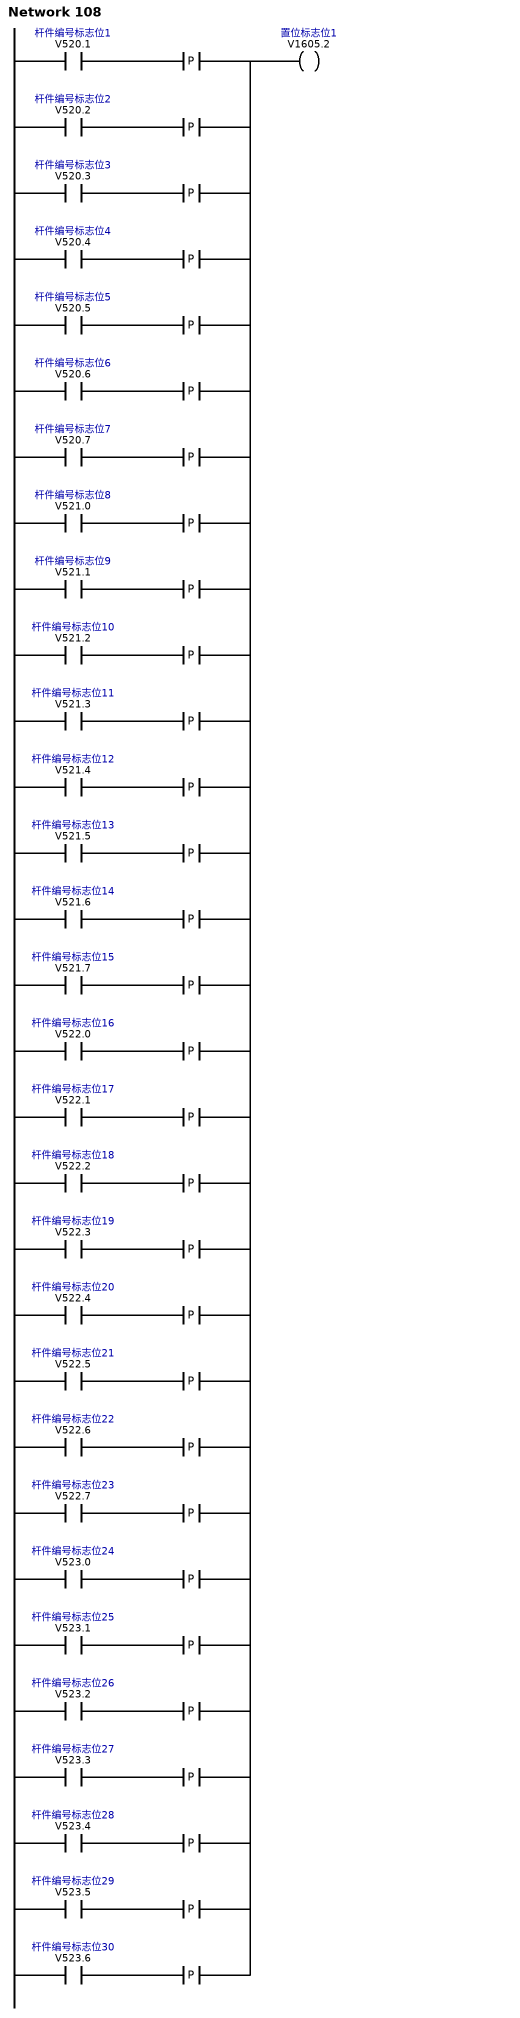
Network 108
LD     杆件编号标志位1:V520.1
EU
LD     杆件编号标志位2:V520.2
EU
OLD
LD     杆件编号标志位3:V520.3
EU
OLD
LD     杆件编号标志位4:V520.4
EU
OLD
LD     杆件编号标志位5:V520.5
EU
OLD
LD     杆件编号标志位6:V520.6
EU
OLD
LD     杆件编号标志位7:V520.7
EU
OLD
LD     杆件编号标志位8:V521.0
EU
OLD
LD     杆件编号标志位9:V521.1
EU
OLD
LD     杆件编号标志位10:V521.2
EU
OLD
LD     杆件编号标志位11:V521.3
EU
OLD
LD     杆件编号标志位12:V521.4
EU
OLD
LD     杆件编号标志位13:V521.5
EU
OLD
LD     杆件编号标志位14:V521.6
EU
OLD
LD     杆件编号标志位15:V521.7
EU
OLD
LD     杆件编号标志位16:V522.0
EU
OLD
LD     杆件编号标志位17:V522.1
EU
OLD
LD     杆件编号标志位18:V522.2
EU
OLD
LD     杆件编号标志位19:V522.3
EU
OLD
LD     杆件编号标志位20:V522.4
EU
OLD
LD     杆件编号标志位21:V522.5
EU
OLD
LD     杆件编号标志位22:V522.6
EU
OLD
LD     杆件编号标志位23:V522.7
EU
OLD
LD     杆件编号标志位24:V523.0
EU
OLD
LD     杆件编号标志位25:V523.1
EU
OLD
LD     杆件编号标志位26:V523.2
EU
OLD
LD     杆件编号标志位27:V523.3
EU
OLD
LD     杆件编号标志位28:V523.4
EU
OLD
LD     杆件编号标志位29:V523.5
EU
OLD
LD     杆件编号标志位30:V523.6
EU
OLD
=      置位标志位1:V1605.2
